// TIA Portal project "sexy pics" (V17)

(* hardware
DEVICE "S7-1200 station_1"  S7-1200 Station
   slot 0: "Rack_0"  S7-1200 Rack  Rack  V1.0
   slot 1: "PLC_1"  CPU 1214C AC/DC/Rly  6ES7 214-1BG40-0XB0  V4.5
DEVICE "HMI_1"  KTP700 Basic PN
   slot 0: "HMI_1"  KTP700 Basic PN  6AV2 123-2GB03-0AX0  17.0.0.0
   slot 1: "HMI_RT_1"  KTP700 Basic PN  6AV2 123-2GB03-0AX0  17.0.0.0
   slot 5: "HMI_1.IE_CP_1"  PROFINET Interface  17.0.0.0
      slot 1: "PROFINET Interface_1"  PROFINET Interface
         slot 1: "Port_1"  Port
*)

// ===== PLC "PLC_1"  CPU 1214C AC/DC/Rly =====

VAR_GLOBAL   // PLC tag table "Default tag table"
   "pbStart" AT %M0.4 : Bool;
   "pbStop" AT %M0.5 : Bool;
   "startTask" AT %M0.0 : Bool;
   "g" AT %M0.1 : Bool;
   "y" AT %M0.2 : Bool;
   "r" AT %M0.3 : Bool;
   "startY" AT %M0.6 : Bool;
   "startR" AT %M0.7 : Bool;
   "reset" AT %M1.0 : Bool;
   "aLow" AT %I0.4 : Bool;
   "aHigh" AT %I0.5 : Bool;
   "wow" AT %M1.1 : Bool;
   "istopper" AT %M1.2 : Bool;
   "digital_In" AT %IW64 : Int;
   "sNorm" AT %MD2 : Real;
   "scaled" AT %MD6 : Real;
   "pbStart2" AT %M1.3 : Bool;
   "pbstop2" AT %M1.4 : Bool;
   "pbStart3" AT %M1.5 : Bool;
   "pbStop3" AT %M1.6 : Bool;
   "halt" AT %M1.7 : Bool;
   "startTask3" AT %M10.0 : Bool;
   "startTask2" AT %M10.1 : Bool;
   "g2" AT %M10.2 : Bool;
   "y2" AT %M10.3 : Bool;
   "r2" AT %M10.4 : Bool;
   "r3" AT %M10.5 : Bool;
   "y3" AT %M10.6 : Bool;
   "inletValveControl" AT %M10.7 : Bool;
   "inletValve" AT %M11.0 : Bool;
   "pbstart5" AT %M11.1 : Bool;
   "pbstop5" AT %M11.2 : Bool;
   "gL" AT %M11.3 : Bool;
   "rR" AT %M11.4 : Bool;
   "yL" AT %M11.5 : Bool;
   "yR" AT %M11.6 : Bool;
   "rL" AT %M11.7 : Bool;
   "gR" AT %M12.0 : Bool;
   "startTask4" AT %M12.1 : Bool;
   "startTask5" AT %M12.2 : Bool;
   "g1" AT %Q0.0 : Bool;
   "y1" AT %Q0.1 : Bool;
   "r1" AT %Q0.2 : Bool;
   "r0" AT %Q0.5 : Bool;
   "y0" AT %Q0.4 : Bool;
   "g0" AT %Q0.3 : Bool;
   "pbStartInput" AT %I0.2 : Bool;
   "pbStartControl" AT %I0.0 : Bool;
   "pbStopControl" AT %I0.1 : Bool;
   "startTaskControl" AT %M12.3 : Bool;
   "aG1" AT %M12.4 : Bool;
   "aY1" AT %M12.5 : Bool;
   "aR1" AT %M12.6 : Bool;
   "aY2" AT %M12.7 : Bool;
   "analogR2" AT %M13.0 : Bool;
   "ag2" AT %M13.1 : Bool;
   "m1Input" AT %MD14 : DInt;
   "m1PT" AT %MD18 : DInt;
   "m1ET" AT %MD22 : DInt;
   "m1CntDown" AT %MD26 : DInt;
   "m1CountUp" AT %MD30 : DInt;
   "m2Input" AT %MD34 : DInt;
   "m2PT" AT %MD38 : DInt;
   "m2ET" AT %MD42 : DInt;
   "m2CntDown" AT %MD46 : DInt;
   "m2CountUp" AT %MD50 : DInt;
   "m3Input" AT %MD54 : DInt;
   "m3PT" AT %MD58 : DInt;
   "m3ET" AT %MD62 : DInt;
   "m3CntDown" AT %MD66 : DInt;
   "m3CountUp" AT %MD70 : DInt;
   "t2_m1Input" AT %MD74 : DInt;
   "t2_m1PT" AT %MD78 : DInt;
   "t2_m1ET" AT %MD82 : DInt;
   "t2_m1CntDown" AT %MD86 : DInt;
   "t2_m1CountUp" AT %MD90 : DInt;
   "t2_m2Input" AT %MD94 : DInt;
   "t2_m2PT" AT %MD98 : DInt;
   "t2_m2ET" AT %MD102 : DInt;
   "t2_m2CntDown" AT %MD106 : DInt;
   "t2_m2CountUp" AT %MD110 : DInt;
   "t2_m3Input" AT %MD114 : DInt;
   "t2_m3PT" AT %MD118 : DInt;
   "t2_m3ET" AT %MD122 : DInt;
   "t2_m3CntDown" AT %MD126 : DInt;
   "t2_m3CountUp" AT %MD130 : DInt;
END_VAR

DATA_BLOCK "Task1_DB"   // DB4
{ S7_Optimized_Access := 'TRUE' }
VERSION : 0.1
// stored: InstanceOfName Task1
"Task1"
BEGIN
END_DATA_BLOCK

DATA_BLOCK "Task1_DB_1"   // DB5
{ S7_Optimized_Access := 'TRUE' }
VERSION : 0.1
// stored: InstanceOfName Task1
"Task1"
BEGIN
END_DATA_BLOCK

DATA_BLOCK "Task1_DB_2"   // DB6
{ S7_Optimized_Access := 'TRUE' }
VERSION : 0.1
// stored: InstanceOfName Task1
"Task1"
BEGIN
END_DATA_BLOCK

DATA_BLOCK "Task2_DB"   // DB8
{ S7_Optimized_Access := 'TRUE' }
VERSION : 0.1
// stored: InstanceOfName Task2
"Task2"
BEGIN
END_DATA_BLOCK

DATA_BLOCK "Task2_DB_1"   // DB9
{ S7_Optimized_Access := 'TRUE' }
VERSION : 0.1
// stored: InstanceOfName Task2
"Task2"
BEGIN
END_DATA_BLOCK

DATA_BLOCK "Task1_DB_3"   // DB10
{ S7_Optimized_Access := 'TRUE' }
VERSION : 0.1
// stored: InstanceOfName Task1
"Task1"
BEGIN
END_DATA_BLOCK

DATA_BLOCK "Task2_DB_2"   // DB11
{ S7_Optimized_Access := 'TRUE' }
VERSION : 0.1
// stored: InstanceOfName Task2
"Task2"
BEGIN
END_DATA_BLOCK

DATA_BLOCK "Task2_DB_3"   // DB12
{ S7_Optimized_Access := 'TRUE' }
VERSION : 0.1
// stored: InstanceOfName Task2
"Task2"
BEGIN
END_DATA_BLOCK

DATA_BLOCK "Task1_DB_4"   // DB17
{ S7_Optimized_Access := 'TRUE' }
VERSION : 0.1
// stored: InstanceOfName Task1
"Task1"
BEGIN
END_DATA_BLOCK

DATA_BLOCK "Task2_DB_4"   // DB18
{ S7_Optimized_Access := 'TRUE' }
VERSION : 0.1
// stored: InstanceOfName Task2
"Task2"
BEGIN
END_DATA_BLOCK

DATA_BLOCK "Task2_DB_5"   // DB19
{ S7_Optimized_Access := 'TRUE' }
VERSION : 0.1
// stored: InstanceOfName Task2
"Task2"
BEGIN
END_DATA_BLOCK

DATA_BLOCK "Task3_DB"   // DB20
{ S7_Optimized_Access := 'TRUE' }
VERSION : 0.1
// stored: InstanceOfName Task3
"Task3"
BEGIN
END_DATA_BLOCK

DATA_BLOCK "task5_DB"   // DB21
{ S7_Optimized_Access := 'TRUE' }
VERSION : 0.1
// stored: InstanceOfName task5
"task5"
BEGIN
END_DATA_BLOCK

DATA_BLOCK "task4_DB"   // DB23
{ S7_Optimized_Access := 'TRUE' }
VERSION : 0.1
// stored: InstanceOfName task4
"task4"
BEGIN
END_DATA_BLOCK

// folder: System blocks/Program resources

DATA_BLOCK "IEC_Timer_0_DB"   // DB1
{ S7_Optimized_Access := 'TRUE' }
AUTHOR : Simatic
FAMILY : IEC
NAME : IEC_TMR
VERSION : 1.0
// stored: InstanceOfName IEC_TIMER
"IEC_TIMER"
BEGIN
END_DATA_BLOCK

DATA_BLOCK "IEC_Timer_0_DB_1"   // DB2
{ S7_Optimized_Access := 'TRUE' }
AUTHOR : Simatic
FAMILY : IEC
NAME : IEC_TMR
VERSION : 1.0
// stored: InstanceOfName IEC_TIMER
"IEC_TIMER"
BEGIN
END_DATA_BLOCK

DATA_BLOCK "IEC_Timer_0_DB_2"   // DB3
{ S7_Optimized_Access := 'TRUE' }
AUTHOR : Simatic
FAMILY : IEC
NAME : IEC_TMR
VERSION : 1.0
// stored: InstanceOfName IEC_TIMER
"IEC_TIMER"
BEGIN
END_DATA_BLOCK

DATA_BLOCK "IEC_Timer_0_DB_3"   // DB7
{ S7_Optimized_Access := 'TRUE' }
AUTHOR : Simatic
FAMILY : IEC
NAME : IEC_TMR
VERSION : 1.0
// stored: InstanceOfName IEC_TIMER
"IEC_TIMER"
BEGIN
END_DATA_BLOCK

DATA_BLOCK "IEC_Timer_0_DB_4"   // DB13
{ S7_Optimized_Access := 'TRUE' }
AUTHOR : Simatic
FAMILY : IEC
NAME : IEC_TMR
VERSION : 1.0
// stored: InstanceOfName IEC_TIMER
"IEC_TIMER"
BEGIN
END_DATA_BLOCK

DATA_BLOCK "LgreenToYellowTimer"   // DB14
{ S7_Optimized_Access := 'TRUE' }
AUTHOR : Simatic
FAMILY : IEC
NAME : IEC_TMR
VERSION : 1.0
// stored: InstanceOfName IEC_TIMER
"IEC_TIMER"
BEGIN
END_DATA_BLOCK

DATA_BLOCK "yellowTimer"   // DB15
{ S7_Optimized_Access := 'TRUE' }
AUTHOR : Simatic
FAMILY : IEC
NAME : IEC_TMR
VERSION : 1.0
// stored: InstanceOfName IEC_TIMER
"IEC_TIMER"
BEGIN
END_DATA_BLOCK

DATA_BLOCK "backToYellowTimer"   // DB16
{ S7_Optimized_Access := 'TRUE' }
AUTHOR : Simatic
FAMILY : IEC
NAME : IEC_TMR
VERSION : 1.0
// stored: InstanceOfName IEC_TIMER
"IEC_TIMER"
BEGIN
END_DATA_BLOCK

DATA_BLOCK "trafficReturnYello"   // DB22
{ S7_Optimized_Access := 'TRUE' }
AUTHOR : Simatic
FAMILY : IEC
NAME : IEC_TMR
VERSION : 1.0
// stored: InstanceOfName IEC_TIMER
"IEC_TIMER"
BEGIN
END_DATA_BLOCK

DATA_BLOCK "IEC_Timer_0_DB_5"   // DB24
{ S7_Optimized_Access := 'TRUE' }
AUTHOR : Simatic
FAMILY : IEC
NAME : IEC_TMR
VERSION : 1.0
// stored: InstanceOfName IEC_TIMER
"IEC_TIMER"
BEGIN
END_DATA_BLOCK

// folder: (top level)

FUNCTION_BLOCK "Task1"   // FB1, LAD
{ S7_Optimized_Access := 'TRUE' }
VERSION : 0.1
   VAR_INPUT
      pbStart : Bool;
      pbStop : Bool;
   END_VAR
   VAR_OUTPUT
      g : Bool;
      r : Bool;
      y : Bool;
      gOut : Bool;
      yOut : Bool;
      rOut : Bool;
   END_VAR
   VAR_TEMP
      m1CountUpddd : DInt;
   END_VAR
BEGIN

REGION Network 1
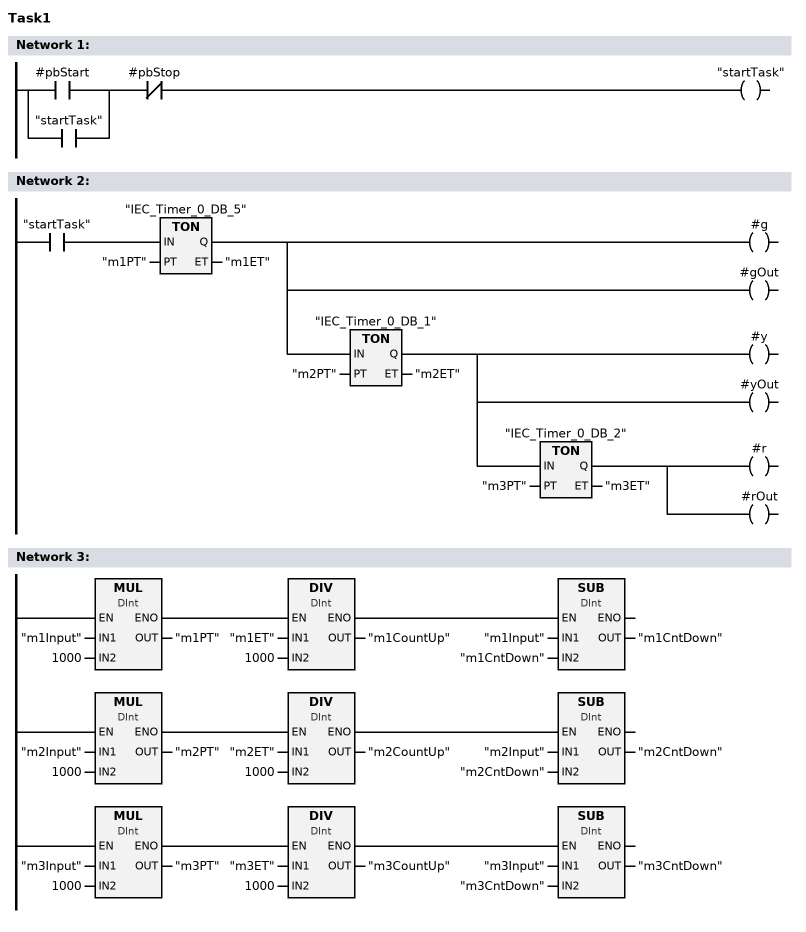
   RUNG wire#powerrail
      Contact( #pbStart )
      wire#w1
      I_Contact( #pbStop )
      Coil( "startTask" )
   END_RUNG
   RUNG wire#powerrail
      Contact( "startTask" )
   END_RUNG wire#w1
   // the same network as SCL:
   "startTask" := (#pbStart OR "startTask") AND NOT #pbStop;
END_REGION

REGION Network 2
   "IEC_Timer_0_DB_5".TON(IN := "startTask", PT := "m1PT", ET => "m1ET");
   #g := "IEC_Timer_0_DB_5".Q;
   #gOut := "IEC_Timer_0_DB_5".Q;
   "IEC_Timer_0_DB_1".TON(IN := "IEC_Timer_0_DB_5".Q, PT := "m2PT", ET => "m2ET");
   #y := "IEC_Timer_0_DB_1".Q;
   #yOut := "IEC_Timer_0_DB_1".Q;
   "IEC_Timer_0_DB_2".TON(IN := "IEC_Timer_0_DB_1".Q, PT := "m3PT", ET => "m3ET");
   #r := "IEC_Timer_0_DB_2".Q;
   #rOut := "IEC_Timer_0_DB_2".Q;
END_REGION

REGION Network 3
   RUNG wire#powerrail
      { S7_Templates := "SrcType := DInt" } Mul(in1 := "m1Input", in2 := 1000, out => "m1PT")
      { S7_Templates := "SrcType := DInt" } Div(in1 := "m1ET", in2 := 1000, out => "m1CountUp")
      { S7_Templates := "SrcType := DInt" } Sub(in1 := "m1Input", in2 := "m1CntDown", out => "m1CntDown")
   END_RUNG
   RUNG wire#powerrail
      { S7_Templates := "SrcType := DInt" } Mul(in1 := "m2Input", in2 := 1000, out => "m2PT")
      { S7_Templates := "SrcType := DInt" } Div(in1 := "m2ET", in2 := 1000, out => "m2CountUp")
      { S7_Templates := "SrcType := DInt" } Sub(in1 := "m2Input", in2 := "m2CntDown", out => "m2CntDown")
   END_RUNG
   RUNG wire#powerrail
      { S7_Templates := "SrcType := DInt" } Mul(in1 := "m3Input", in2 := 1000, out => "m3PT")
      { S7_Templates := "SrcType := DInt" } Div(in1 := "m3ET", in2 := 1000, out => "m3CountUp")
      { S7_Templates := "SrcType := DInt" } Sub(in1 := "m3Input", in2 := "m3CntDown", out => "m3CntDown")
   END_RUNG
   // the same network as SCL:
   "m1PT" := "m1Input" * 1000;
   "m1CountUp" := "m1ET" / 1000;
   "m1CntDown" := "m1Input" - "m1CntDown";
   "m2PT" := "m2Input" * 1000;
   "m2CountUp" := "m2ET" / 1000;
   "m2CntDown" := "m2Input" - "m2CntDown";
   "m3PT" := "m3Input" * 1000;
   "m3CountUp" := "m3ET" / 1000;
   "m3CntDown" := "m3Input" - "m3CntDown";
END_REGION
END_FUNCTION_BLOCK

FUNCTION_BLOCK "Task2"   // FB2, LAD
{ S7_Optimized_Access := 'TRUE' }
VERSION : 0.1
   VAR_INPUT
      pbStart2 : Bool;
      pbStop2 : Bool;
   END_VAR
   VAR_OUTPUT
      g2 : Bool;
      y2 : Bool;
      r2 : Bool;
      yOut : Bool;
      rOut : Bool;
      gOut : Bool;
   END_VAR
   VAR_TEMP   // added for the SCL form of the ladder/FBD networks
      _w1 : Bool;
   END_VAR
BEGIN

REGION Network 1
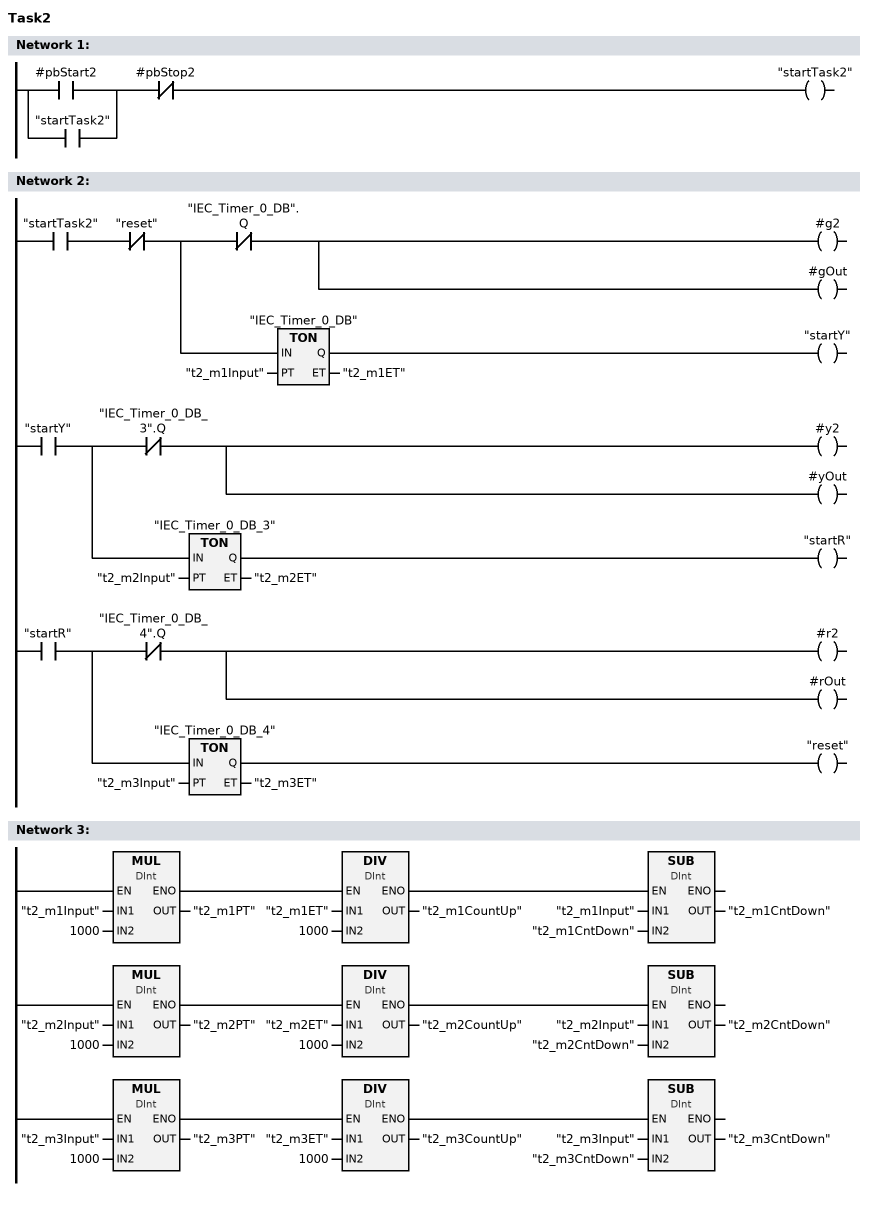
   RUNG wire#powerrail
      Contact( #pbStart2 )
      wire#w1
      I_Contact( #pbStop2 )
      Coil( "startTask2" )
   END_RUNG
   RUNG wire#powerrail
      Contact( "startTask2" )
   END_RUNG wire#w1
   // the same network as SCL:
   "startTask2" := (#pbStart2 OR "startTask2") AND NOT #pbStop2;
END_REGION

REGION Network 2
   #_w1 := "startTask2" AND NOT "reset";
   #g2 := #_w1 AND NOT "IEC_Timer_0_DB".Q;
   #gOut := #g2;
   "IEC_Timer_0_DB".TON(IN := #_w1, PT := "t2_m1Input", ET => "t2_m1ET");
   "startY" := "IEC_Timer_0_DB".Q;
   #y2 := "startY" AND NOT "IEC_Timer_0_DB_3".Q;
   #yOut := #y2;
   "IEC_Timer_0_DB_3".TON(IN := "startY", PT := "t2_m2Input", ET => "t2_m2ET");
   "startR" := "IEC_Timer_0_DB_3".Q;
   #r2 := "startR" AND NOT "IEC_Timer_0_DB_4".Q;
   #rOut := #r2;
   "IEC_Timer_0_DB_4".TON(IN := "startR", PT := "t2_m3Input", ET => "t2_m3ET");
   "reset" := "IEC_Timer_0_DB_4".Q;
END_REGION

REGION Network 3
   RUNG wire#powerrail
      { S7_Templates := "SrcType := DInt" } Mul(in1 := "t2_m1Input", in2 := 1000, out => "t2_m1PT")
      { S7_Templates := "SrcType := DInt" } Div(in1 := "t2_m1ET", in2 := 1000, out => "t2_m1CountUp")
      { S7_Templates := "SrcType := DInt" } Sub(in1 := "t2_m1Input", in2 := "t2_m1CntDown", out => "t2_m1CntDown")
   END_RUNG
   RUNG wire#powerrail
      { S7_Templates := "SrcType := DInt" } Mul(in1 := "t2_m2Input", in2 := 1000, out => "t2_m2PT")
      { S7_Templates := "SrcType := DInt" } Div(in1 := "t2_m2ET", in2 := 1000, out => "t2_m2CountUp")
      { S7_Templates := "SrcType := DInt" } Sub(in1 := "t2_m2Input", in2 := "t2_m2CntDown", out => "t2_m2CntDown")
   END_RUNG
   RUNG wire#powerrail
      { S7_Templates := "SrcType := DInt" } Mul(in1 := "t2_m3Input", in2 := 1000, out => "t2_m3PT")
      { S7_Templates := "SrcType := DInt" } Div(in1 := "t2_m3ET", in2 := 1000, out => "t2_m3CountUp")
      { S7_Templates := "SrcType := DInt" } Sub(in1 := "t2_m3Input", in2 := "t2_m3CntDown", out => "t2_m3CntDown")
   END_RUNG
   // the same network as SCL:
   "t2_m1PT" := "t2_m1Input" * 1000;
   "t2_m1CountUp" := "t2_m1ET" / 1000;
   "t2_m1CntDown" := "t2_m1Input" - "t2_m1CntDown";
   "t2_m2PT" := "t2_m2Input" * 1000;
   "t2_m2CountUp" := "t2_m2ET" / 1000;
   "t2_m2CntDown" := "t2_m2Input" - "t2_m2CntDown";
   "t2_m3PT" := "t2_m3Input" * 1000;
   "t2_m3CountUp" := "t2_m3ET" / 1000;
   "t2_m3CntDown" := "t2_m3Input" - "t2_m3CntDown";
END_REGION
END_FUNCTION_BLOCK

FUNCTION_BLOCK "Task3"   // FB3, LAD
{ S7_Optimized_Access := 'TRUE' }
VERSION : 0.1
   VAR_INPUT
      pbStart3 : Bool;
      pbStop3 : Bool;
      inletValveControl : Bool;
      buttonLow3 : Bool;
   END_VAR
   VAR_OUTPUT
      LLS : Bool;
      inletValve : Bool;
      y3 : Bool;
   END_VAR
   VAR
      Memstarter : Bool;
      Memstopper : Bool;
   END_VAR
BEGIN

REGION Network 1
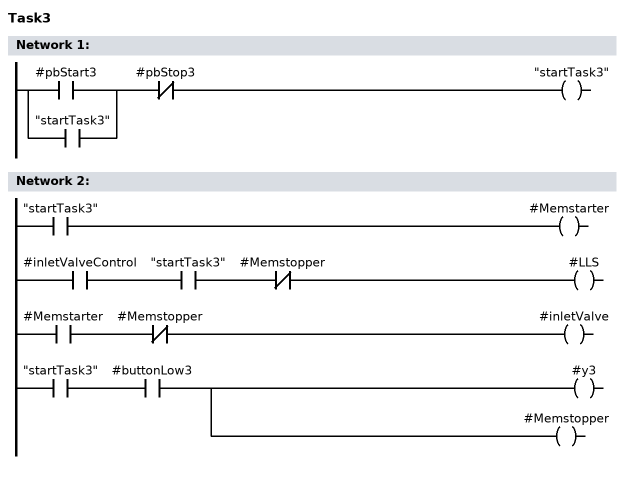
   RUNG wire#powerrail
      Contact( #pbStart3 )
      wire#w1
      I_Contact( #pbStop3 )
      Coil( "startTask3" )
   END_RUNG
   RUNG wire#powerrail
      Contact( "startTask3" )
   END_RUNG wire#w1
   // the same network as SCL:
   "startTask3" := (#pbStart3 OR "startTask3") AND NOT #pbStop3;
END_REGION

REGION Network 2
   RUNG wire#powerrail
      Contact( "startTask3" )
      Coil( #Memstarter )
   END_RUNG
   RUNG wire#powerrail
      Contact( #inletValveControl )
      Contact( "startTask3" )
      I_Contact( #Memstopper )
      Coil( #LLS )
   END_RUNG
   RUNG wire#powerrail
      Contact( #Memstarter )
      I_Contact( #Memstopper )
      Coil( #inletValve )
   END_RUNG
   RUNG wire#powerrail
      Contact( "startTask3" )
      Contact( #buttonLow3 )
      wire#w1
      Coil( #y3 )
   END_RUNG
   RUNG wire#w1
      Coil( #Memstopper )
   END_RUNG
   // the same network as SCL:
   #Memstarter := "startTask3";
   #LLS := #inletValveControl AND "startTask3" AND NOT #Memstopper;
   #inletValve := #Memstarter AND NOT #Memstopper;
   #y3 := "startTask3" AND #buttonLow3;
   #Memstopper := #y3;
END_REGION
END_FUNCTION_BLOCK

FUNCTION_BLOCK "task4"   // FB4, LAD
{ S7_Optimized_Access := 'TRUE' }
VERSION : 0.1
   VAR_INPUT
      pbStart : Bool;
      pbStop : Bool;
   END_VAR
   VAR_OUTPUT
      r : Bool;
      y : Bool;
      g : Bool;
   END_VAR
   VAR_TEMP   // added for the SCL form of the ladder/FBD networks
      _w1 : Bool;
   END_VAR
BEGIN

REGION Network 1
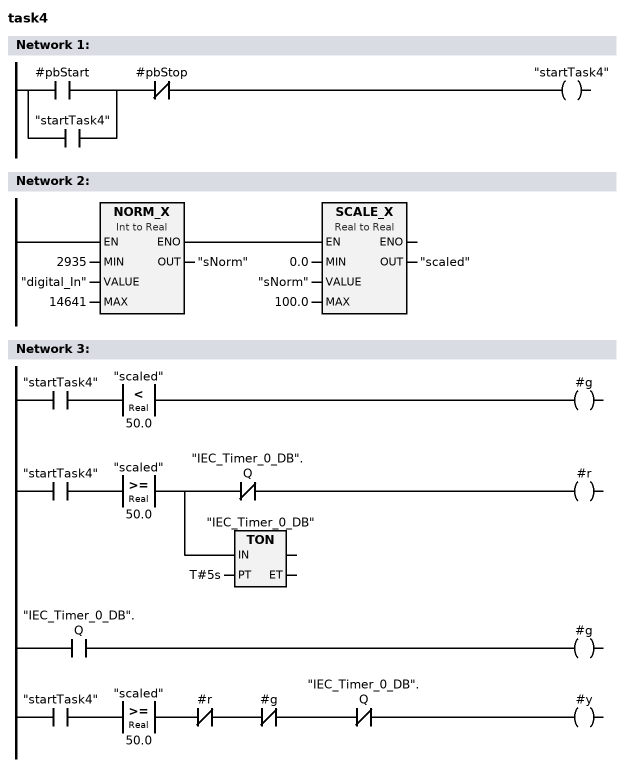
   RUNG wire#powerrail
      Contact( #pbStart )
      wire#w1
      I_Contact( #pbStop )
      Coil( "startTask4" )
   END_RUNG
   RUNG wire#powerrail
      Contact( "startTask4" )
   END_RUNG wire#w1
   // the same network as SCL:
   "startTask4" := (#pbStart OR "startTask4") AND NOT #pbStop;
END_REGION

REGION Network 2
   RUNG wire#powerrail
      { S7_Templates := "[SrcType := Int, DestType := Real]" } Normalize(min := 2935, value := "digital_In", max := 14641, out => "sNorm")
      { S7_Templates := "[SrcType := Real, DestType := Real]" } Scale(min := 0.0, value := "sNorm", max := 100.0, out => "scaled")
   END_RUNG
   // the same network as SCL:
   "sNorm" := NORM_X(MIN := 2935, VALUE := "digital_In", MAX := 14641);
   "scaled" := SCALE_X(MIN := 0.0, VALUE := "sNorm", MAX := 100.0);
END_REGION

REGION Network 3
   #g := "startTask4" AND ("scaled" < 50.0);
   #_w1 := "startTask4" AND ("scaled" >= 50.0);
   #r := #_w1 AND NOT "IEC_Timer_0_DB".Q;
   "IEC_Timer_0_DB".TON(IN := #_w1, PT := T#5s);
   #g := "IEC_Timer_0_DB".Q;
   #y := "startTask4" AND ("scaled" >= 50.0) AND NOT #r AND NOT #g AND NOT "IEC_Timer_0_DB".Q;
END_REGION
END_FUNCTION_BLOCK

FUNCTION_BLOCK "task5"   // FB5, LAD
{ S7_Optimized_Access := 'TRUE' }
VERSION : 0.1
   VAR_INPUT
      pbStart : Bool;
      pbStop : Bool;
   END_VAR
   VAR_OUTPUT
      gL : Bool;
      rR : Bool;
      yL : Bool;
      yR : Bool;
      rL : Bool;
      gR : Bool;
      analog_yL : Bool;
      analog_yR : Bool;
      analog_gL : Bool;
      analog_gR : Bool;
      analog_rL : Bool;
      analog_rR : Bool;
   END_VAR
   VAR
      interlockReturn : Bool;
      toYellow : Bool;
      interlockStopperYellow : Bool;
      returnBackToYellow : Bool;
   END_VAR
   VAR_TEMP   // added for the SCL form of the ladder/FBD networks
      _w1 : Bool;
   END_VAR
BEGIN

REGION Network 1
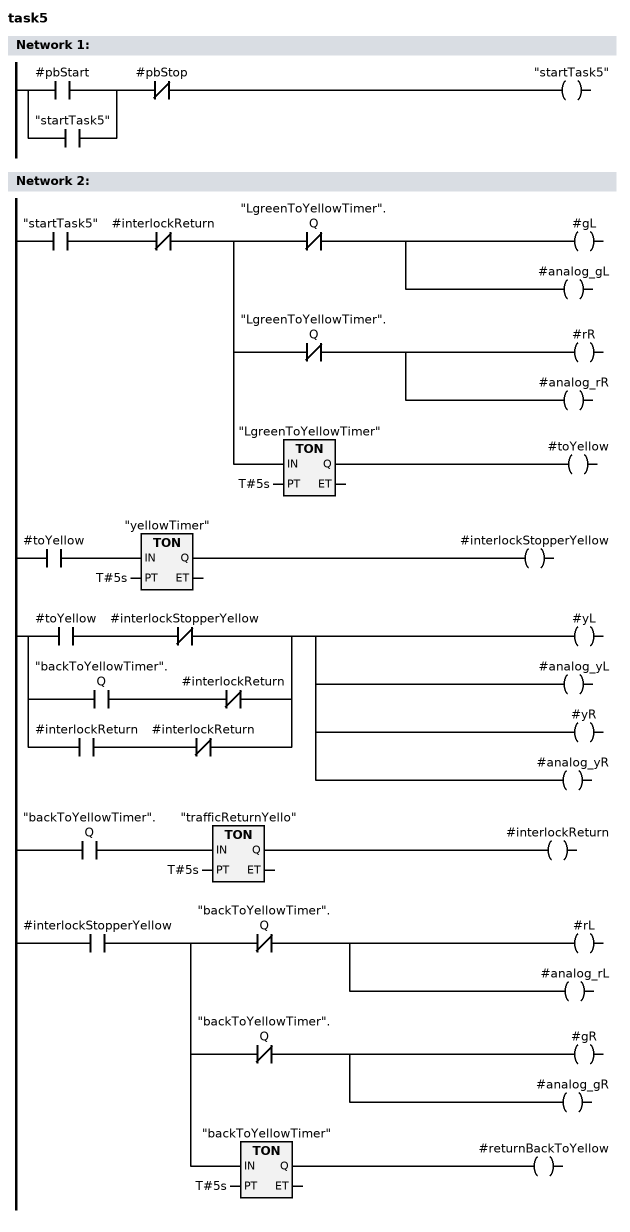
   RUNG wire#powerrail
      Contact( #pbStart )
      wire#w1
      I_Contact( #pbStop )
      Coil( "startTask5" )
   END_RUNG
   RUNG wire#powerrail
      Contact( "startTask5" )
   END_RUNG wire#w1
   // the same network as SCL:
   "startTask5" := (#pbStart OR "startTask5") AND NOT #pbStop;
END_REGION

REGION Network 2
   #_w1 := "startTask5" AND NOT #interlockReturn;
   #gL := #_w1 AND NOT "LgreenToYellowTimer".Q;
   #analog_gL := #gL;
   #rR := #_w1 AND NOT "LgreenToYellowTimer".Q;
   #analog_rR := #rR;
   "LgreenToYellowTimer".TON(IN := #_w1, PT := T#5s);
   #toYellow := "LgreenToYellowTimer".Q;
   "yellowTimer".TON(IN := #toYellow, PT := T#5s);
   #interlockStopperYellow := "yellowTimer".Q;
   #yL := (#toYellow AND NOT #interlockStopperYellow) OR ("backToYellowTimer".Q AND NOT #interlockReturn) OR (#interlockReturn AND NOT #interlockReturn);
   #analog_yL := #yL;
   #yR := #yL;
   #analog_yR := #yL;
   "trafficReturnYello".TON(IN := "backToYellowTimer".Q, PT := T#5s);
   #interlockReturn := "trafficReturnYello".Q;
   #rL := #interlockStopperYellow AND NOT "backToYellowTimer".Q;
   #analog_rL := #rL;
   #gR := #interlockStopperYellow AND NOT "backToYellowTimer".Q;
   #analog_gR := #gR;
   "backToYellowTimer".TON(IN := #interlockStopperYellow, PT := T#5s);
   #returnBackToYellow := "backToYellowTimer".Q;
END_REGION
END_FUNCTION_BLOCK

ORGANIZATION_BLOCK "Main"   // OB1, LAD, ProgramCycle
TITLE = "Main Program Sweep (Cycle)"
{ S7_Optimized_Access := 'TRUE' }
VERSION : 0.1
   VAR_INPUT
      Initial_Call : Bool;   // Initial call of this OB
      Remanence : Bool;   // =True, if remanent data are available
   END_VAR
BEGIN

REGION Network 1
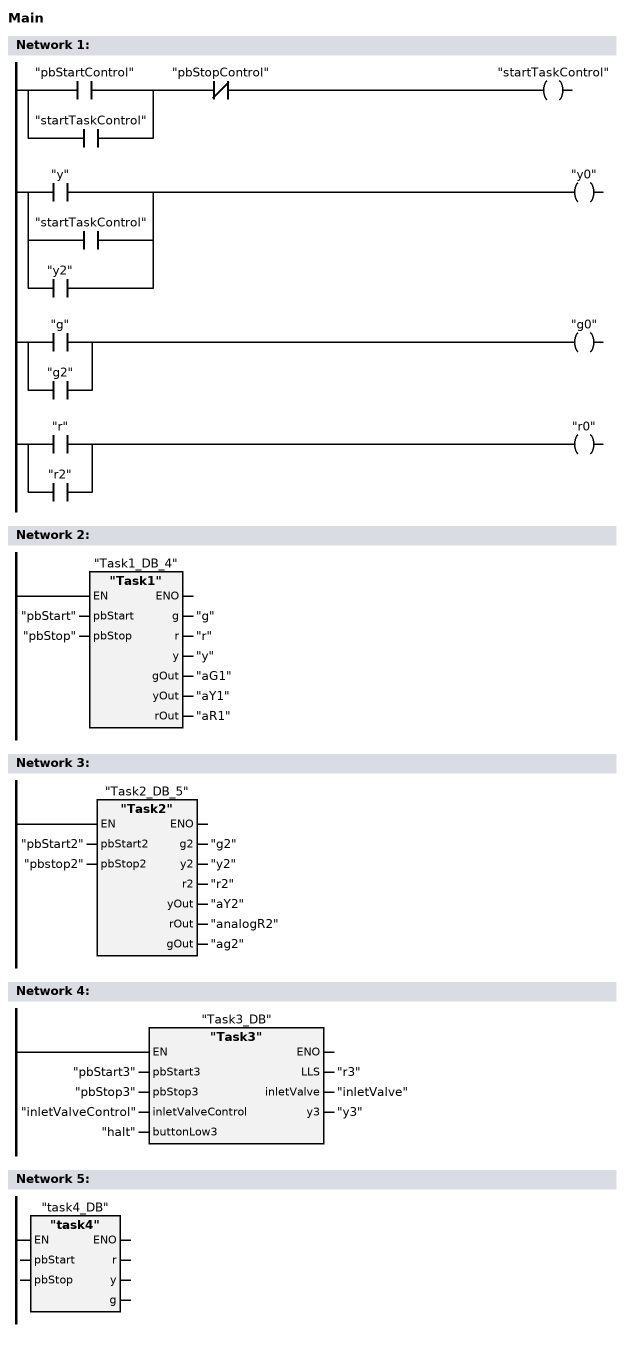
   RUNG wire#powerrail
      Contact( "pbStartControl" )
      wire#w1
      I_Contact( "pbStopControl" )
      Coil( "startTaskControl" )
   END_RUNG
   RUNG wire#powerrail
      Contact( "startTaskControl" )
   END_RUNG wire#w1
   RUNG wire#powerrail
      Contact( "y" )
      wire#w2
      Coil( "y0" )
   END_RUNG
   RUNG wire#powerrail
      Contact( "startTaskControl" )
   END_RUNG wire#w2
   RUNG wire#powerrail
      Contact( "y2" )
   END_RUNG wire#w2
   RUNG wire#powerrail
      Contact( "g" )
      wire#w3
      Coil( "g0" )
   END_RUNG
   RUNG wire#powerrail
      Contact( "g2" )
   END_RUNG wire#w3
   RUNG wire#powerrail
      Contact( "r" )
      wire#w4
      Coil( "r0" )
   END_RUNG
   RUNG wire#powerrail
      Contact( "r2" )
   END_RUNG wire#w4
   // the same network as SCL:
   "startTaskControl" := ("pbStartControl" OR "startTaskControl") AND NOT "pbStopControl";
   "y0" := "y" OR "startTaskControl" OR "y2";
   "g0" := "g" OR "g2";
   "r0" := "r" OR "r2";
END_REGION

REGION Network 2
   RUNG wire#powerrail
      "Task1_DB_4"(pbStart := "pbStart", pbStop := "pbStop", g => "g", r => "r", y => "y", gOut => "aG1", yOut => "aY1", rOut => "aR1")
   END_RUNG
   // the same network as SCL:
   "Task1_DB_4"(pbStart := "pbStart",   // "Task1"
                pbStop := "pbStop",
                g => "g",
                r => "r",
                y => "y",
                gOut => "aG1",
                yOut => "aY1",
                rOut => "aR1");
END_REGION

REGION Network 3
   RUNG wire#powerrail
      "Task2_DB_5"(pbStart2 := "pbStart2", pbStop2 := "pbstop2", g2 => "g2", y2 => "y2", r2 => "r2", yOut => "aY2", rOut => "analogR2", gOut => "ag2")
   END_RUNG
   // the same network as SCL:
   "Task2_DB_5"(pbStart2 := "pbStart2",   // "Task2"
                pbStop2 := "pbstop2",
                g2 => "g2",
                y2 => "y2",
                r2 => "r2",
                yOut => "aY2",
                rOut => "analogR2",
                gOut => "ag2");
END_REGION

REGION Network 4
   RUNG wire#powerrail
      "Task3_DB"(pbStart3 := "pbStart3", pbStop3 := "pbStop3", inletValveControl := "inletValveControl", buttonLow3 := "halt", LLS => "r3", inletValve => "inletValve", y3 => "y3")
   END_RUNG
   // the same network as SCL:
   "Task3_DB"(pbStart3 := "pbStart3",   // "Task3"
              pbStop3 := "pbStop3",
              inletValveControl := "inletValveControl",
              buttonLow3 := "halt",
              LLS => "r3",
              inletValve => "inletValve",
              y3 => "y3");
END_REGION

REGION Network 5
   RUNG wire#powerrail
      "task4_DB"(pbStart :=, pbStop :=, r =>, y =>, g =>)
   END_RUNG
   // the same network as SCL:
   "task4_DB"();   // "task4"
END_REGION
END_ORGANIZATION_BLOCK

(* ===== HMI "HMI_RT_1" =====
system functions are stored by id; their names below are inferred from use
connection "HMI_Connection_1": ETHERNET, SMART_S7_1200_OMS

HMI tags "Default tag table"
   "pbStart" : Bool = PLC pbStart AT %M0.4, 1 s
   "pbStop" : Bool = PLC pbStop AT %M0.5, 1 s
   "g" : Bool = PLC g AT %M0.1, 1 s
   "y" : Bool = PLC y AT %M0.2, 1 s
   "r" : Bool = PLC r AT %M0.3, 1 s
   "pbStart2" : Bool = PLC pbStart2 AT %M1.3, 1 s
   "halt" : Bool = PLC halt AT %M1.7, 1 s
   "pbStart3" : Bool = PLC pbStart3 AT %M1.5, 1 s
   "pbStop3" : Bool = PLC pbStop3 AT %M1.6, 1 s
   "pbstop2" : Bool = PLC pbstop2 AT %M1.4, 1 s
   "g2" : Bool = PLC g2 AT %M10.2, 1 s
   "y2" : Bool = PLC y2 AT %M10.3, 1 s
   "r3" : Bool = PLC r3 AT %M10.5, 1 s
   "y3" : Bool = PLC y3 AT %M10.6, 1 s
   "inletValve" : Bool = PLC inletValve AT %M11.0, 1 s
   "r2" : Bool = PLC r2 AT %M10.4, 1 s
   "yL" : Bool = PLC yL AT %M11.5, 1 s
   "gL" : Bool = PLC gL AT %M11.3, 1 s
   "rL" : Bool = PLC rL AT %M11.7, 1 s
   "rR" : Bool = PLC rR AT %M11.4, 1 s
   "yR" : Bool = PLC yR AT %M11.6, 1 s
   "gR" : Bool = PLC gR AT %M12.0, 1 s
   "aHigh" : Bool = PLC aHigh AT %I0.5, 1 s
   "pbstart5" : Bool = PLC pbstart5 AT %M11.1, 1 s
   "pbstop5" : Bool = PLC pbstop5 AT %M11.2, 1 s
   "m1Input" : DInt = PLC m1Input AT %MD14, 1 s
   "m2Input" : DInt = PLC m2Input AT %MD34, 1 s
   "m1CntDown" : DInt = PLC m1CntDown AT %MD26, 1 s
   "m1CountUp" : DInt = PLC m1CountUp AT %MD30, 1 s
   "m2CntDown" : DInt = PLC m2CntDown AT %MD46, 1 s
   "m2CountUp" : DInt = PLC m2CountUp AT %MD50, 1 s
   "m3Input" : DInt = PLC m3Input AT %MD54, 1 s
   "m3CntDown" : DInt = PLC m3CntDown AT %MD66, 1 s
   "m3CountUp" : DInt = PLC m3CountUp AT %MD70, 1 s
   "t2_m1Input" : DInt = PLC t2_m1Input AT %MD74, 1 s
   "t2_m2Input" : DInt = PLC t2_m2Input AT %MD94, 1 s
   "t2_m3Input" : DInt = PLC t2_m3Input AT %MD114, 1 s
   "t2_m1CntDown" : DInt = PLC t2_m1CntDown AT %MD86, 1 s
   "t2_m1CountUp" : DInt = PLC t2_m1CountUp AT %MD90, 1 s
   "t2_m2CntDown" : DInt = PLC t2_m2CntDown AT %MD106, 1 s
   "t2_m2CountUp" : DInt = PLC t2_m2CountUp AT %MD110, 1 s
   "t2_m3CntDown" : DInt = PLC t2_m3CntDown AT %MD126, 1 s
   "t2_m3CountUp" : DInt = PLC t2_m3CountUp AT %MD130, 1 s
   "scaled" : Real = PLC scaled AT %MD6, 1 s

screen "Root screen" 800x480, template "Template_1"
   GraphicView "Graphic view_1" at 18,20 size 84x84; Picture "275542019_5352027011475781_8646763153125628757_n"
   TextField "Text field_1" at 111,20 size 617x37; Text 'PLC TRAINING COMPILATION OF PROJECTS'
   TextField "Text field_2" at 111,64 size 173x25; Text 'BY: NICO GUARNES'
   Button "Button_1" at 54,156 size 212x100; TextOff 'PRACTICAL 1: Motor Control'
      on Release: ActivateScreen("Practical_1", 0)
   Button "Button_2" at 299,156 size 212x100; TextOff 'PRACTICAL 2: Sequential Motor Control'
      on Release: ActivateScreen("Practical_2", 0)
   Button "Button_3" at 546,156 size 212x100; TextOff 'PRACTICAL 3: Control Level of a Single Tank'
      on Release: ActivateScreen("Practical_3", 0)
   Button "Button_4" at 50,290 size 212x100; TextOff 'PRACTICAL 4: Control Mixing in a Tank'
      on Release: ActivateScreen("Practical_4", 0)
   Button "Button_5" at 299,290 size 212x100; TextOff 'PRACTICAL 5: Traffic Lights'
      on Release: ActivateScreen("Practical_5", 0)

screen "Practical_1" 800x480, template "Template_1"
   GraphicView "Graphic view_1" at 18,20 size 84x84; Picture "275542019_5352027011475781_8646763153125628757_n"
   TextField "Text field_1" at 111,20 size 455x37; Text 'PRACTICAL 1 : MOTOR CONTROL'
   TextField "Text field_2" at 111,64 size 173x25; Text 'BY: NICO GUARNES'
   Button "Button_1" at 715,41 size 54x48; TextOff 'Text'; PictureOff "home_64dp_FFBE33_FILL1_wght400_GRAD0_opsz48"
      on Release: ActivateScreen("Root screen", 0); ResetBit("pbStop")
      on Press: SetBit("pbStop")
   Button "Button_2" at 11,431 size 96x32; TextOff 'START'
      on Release: ResetBit("pbStart")
      on Press: SetBit("pbStart")
   Button "Button_3" at 123,431 size 96x32; TextOff 'STOP'
      on Press: SetBit("pbStop")
      on Release: ResetBit("pbStop")
   GraphicView "Graphic view_2" at 58,159 size 187x105; Picture "Graphic_3"
      Visibility <- "g"
   GraphicView "Graphic view_3" at 58,159 size 187x105; Picture "Graphic_4"
      Visibility <- "g"
   GraphicView "Graphic view_4" at 308,161 size 187x105; Picture "Graphic_3"
      Visibility <- "y"
   GraphicView "Graphic view_6" at 540,161 size 187x105; Picture "Graphic_3"
      Visibility <- "r"
   GraphicView "Graphic view_5" at 308,161 size 187x105; Picture "Graphic_5"
      Visibility <- "y"
   GraphicView "Graphic view_7" at 540,161 size 187x105; Picture "Graphic_6"
      Visibility <- "r"
   TextField "Text field_11" at 64,138 size 56x17; Text 'MOTOR 1'
   TextField "Text field_3" at 322,134 size 56x17; Text 'MOTOR 1'
   TextField "Text field_4" at 580,130 size 56x17; Text 'MOTOR 3'
   IOField "I/O field_1" at 69,282 size 96x32; FormatPattern 999
      ProcessValue <- "m1Input"
   IOField "I/O field_4" at 69,324 size 96x32; FormatPattern 999
      ProcessValue <- "m1CntDown"
   IOField "I/O field_5" at 69,366 size 96x32; FormatPattern 999
      ProcessValue <- "m1CountUp"
   IOField "I/O field_2" at 323,282 size 96x32; FormatPattern 999
      ProcessValue <- "m2Input"
   IOField "I/O field_3" at 323,324 size 96x32; FormatPattern 999
      ProcessValue <- "m2CntDown"
   IOField "I/O field_6" at 323,366 size 96x32; FormatPattern 999
      ProcessValue <- "m2CountUp"
   IOField "I/O field_7" at 563,282 size 96x32; FormatPattern 999
      ProcessValue <- "m3Input"
   IOField "I/O field_8" at 563,324 size 96x32; FormatPattern 999
      ProcessValue <- "m3CntDown"
   IOField "I/O field_9" at 563,366 size 96x32; FormatPattern 999
      ProcessValue <- "m3CountUp"
   TextField "Text field_5" at 168,332 size 72x17; Text 'Count Down'
   TextField "Text field_6" at 167,373 size 56x17; Text 'Count Up'
   TextField "Text field_7" at 172,290 size 92x17; Text 'Preset Time (s)'
   TextField "Text field_8" at 422,332 size 72x17; Text 'Count Down'
   TextField "Text field_9" at 421,373 size 56x17; Text 'Count Up'
   TextField "Text field_10" at 426,290 size 92x17; Text 'Preset Time (s)'
   TextField "Text field_12" at 676,332 size 72x17; Text 'Count Down'
   TextField "Text field_13" at 675,373 size 56x17; Text 'Count Up'
   TextField "Text field_14" at 680,290 size 92x17; Text 'Preset Time (s)'

screen "Practical_2" 800x480, template "Template_1"
   GraphicView "Graphic view_1" at 18,20 size 84x84; Picture "275542019_5352027011475781_8646763153125628757_n"
   TextField "Text field_1" at 111,20 size 582x34; Text 'PRACTICAL 2 : SEQUENTIAL MOTOR CONTROL'
   TextField "Text field_2" at 111,56 size 173x25; Text 'BY: NICO GUARNES'
   Button "Button_1" at 715,41 size 54x48; TextOff 'Text'; PictureOff "home_64dp_FFBE33_FILL1_wght400_GRAD0_opsz48"
      on Release: ActivateScreen("Root screen", 0); ResetBit("pbstop2")
      on Press: SetBit("pbstop2")
   Button "Button_2" at 11,431 size 96x32; TextOff 'START'
      on Release: ResetBit("pbStart2")
      on Press: SetBit("pbStart2")
   Button "Button_3" at 123,431 size 96x32; TextOff 'STOP'
      on Release: ResetBit("pbstop2")
      on Press: SetBit("pbstop2")
   GraphicView "Graphic view_2" at 58,181 size 187x105; Picture "Graphic_3"
   GraphicView "Graphic view_3" at 58,181 size 187x105; Picture "Graphic_4"
      Visibility <- "g2"
   GraphicView "Graphic view_4" at 280,181 size 187x105; Picture "Graphic_3"
   GraphicView "Graphic view_6" at 518,188 size 187x105; Picture "Graphic_3"
   GraphicView "Graphic view_5" at 280,181 size 187x105; Picture "Graphic_5"
      Visibility <- "y2"
   GraphicView "Graphic view_7" at 518,188 size 187x105; Picture "Graphic_6"
      Visibility <- "r2"
   TextField "Text field_11" at 64,156 size 56x17; Text 'MOTOR 1'
   TextField "Text field_3" at 280,156 size 56x17; Text 'MOTOR 2'
   TextField "Text field_4" at 518,163 size 56x17; Text 'MOTOR 3'
   IOField "I/O field_1" at 65,310 size 96x32; FormatPattern 999
      ProcessValue <- "t2_m1Input"
   IOField "I/O field_4" at 65,352 size 96x32; FormatPattern 999
      ProcessValue <- "t2_m1CntDown"
   IOField "I/O field_5" at 65,394 size 96x32; FormatPattern 999
      ProcessValue <- "t2_m1CountUp"
   IOField "I/O field_2" at 295,310 size 96x32; FormatPattern 999
      ProcessValue <- "t2_m2Input"
   IOField "I/O field_3" at 295,352 size 96x32; FormatPattern 999
      ProcessValue <- "t2_m2CntDown"
   IOField "I/O field_6" at 295,394 size 96x32; FormatPattern 999
      ProcessValue <- "t2_m2CountUp"
   IOField "I/O field_7" at 525,310 size 96x32; FormatPattern 999
      ProcessValue <- "t2_m3Input"
   IOField "I/O field_8" at 525,352 size 96x32; FormatPattern 999
      ProcessValue <- "t2_m3CntDown"
   IOField "I/O field_9" at 525,394 size 96x32; FormatPattern 999
      ProcessValue <- "t2_m3CountUp"
   TextField "Text field_5" at 166,361 size 72x17; Text 'Count Down'
   TextField "Text field_6" at 165,402 size 56x17; Text 'Count Up'
   TextField "Text field_7" at 170,319 size 92x17; Text 'Preset Time (s)'
   TextField "Text field_8" at 402,361 size 72x17; Text 'Count Down'
   TextField "Text field_9" at 403,402 size 56x17; Text 'Count Up'
   TextField "Text field_10" at 402,319 size 92x17; Text 'Preset Time (s)'
   TextField "Text field_12" at 628,361 size 72x17; Text 'Count Down'
   TextField "Text field_13" at 625,402 size 56x17; Text 'Count Up'
   TextField "Text field_14" at 626,319 size 92x17; Text 'Preset Time (s)'

screen "Practical_3" 800x480, template "Template_1"
   GraphicView "Graphic view_1" at 18,20 size 84x84; Picture "275542019_5352027011475781_8646763153125628757_n"
   TextField "Text field_1" at 111,20 size 574x34; Text 'PRACTICAL 3 : SINGLE TANK CONTROL LEVEL'
   TextField "Text field_2" at 111,64 size 173x25; Text 'BY: NICO GUARNES'
   Button "Button_1" at 715,41 size 54x48; TextOff 'Text'; PictureOff "home_64dp_FFBE33_FILL1_wght400_GRAD0_opsz48"
      on Release: ActivateScreen("Root screen", 0)
   Button "Button_2" at 15,151 size 96x32; TextOff 'START'
      on Release: ResetBit("pbStart3")
      on Press: SetBit("pbStart3")
   Button "Button_3" at 15,203 size 96x32; TextOff 'STOP'
      on Release: ResetBit("pbStop3")
      on Press: SetBit("pbStop3")
   GraphicView "Graphic view_5" at 497,432 size 125x38; Picture "Graphic_13"
   GraphicView "Graphic view_10" at 464,432 size 34x38; Picture "Graphic_21"
   GraphicView "Graphic view_9" at 464,397 size 34x38; Picture "Graphic_18"
   GraphicView "Graphic view_4" at 222,144 size 126x34; Picture "Graphic_13"
   GraphicView "Graphic view_6" at 243,140 size 43x36; Picture "Graphic_19"
   GraphicView "Graphic view_2" at 344,143 size 39x36; Picture "Graphic_16"
   GraphicView "Graphic view_8" at 345,177 size 38x55; Picture "Graphic_18"
   GraphicView "Graphic view_7" at 547,431 size 43x36; Picture "Graphic_19"
   GraphicView "Graphic view_3" at 332,203 size 190x208; Picture "Graphic_11"
   Circle "Circle_1" at 351,226 size 25x25
      Appearance <- "y3"
   Circle "Circle_2" at 356,368 size 25x25
      Appearance <- "r3"
   TextField "Text field_3" at 292,227 size 38x25; Text 'LLH'
   TextField "Text field_4" at 297,367 size 36x25; Text 'LLS'
   GraphicView "Graphic view_11" at 244,140 size 43x36; Picture "Graphic_22"
      Visibility <- "inletValve"
   GraphicView "Graphic view_12" at 547,431 size 43x36; Picture "Graphic_23"
      Visibility <- "y3"
   TextField "Text field_11" at 544,414 size 84x17; Text 'OUTLET VALVE'
   TextField "Text field_5" at 222,124 size 73x17; Text 'INLET VALVE'
   Bar "Bar_1" at 206,203 size 80x212; MinimumValue 0; MaximumValue 100

screen "Practical_4" 800x480, template "Template_1"
   GraphicView "Graphic view_16" at 409,434 size 97x26; Picture "Graphic_13"
   GraphicView "Graphic view_17" at 465,431 size 33x28; Picture "Graphic_19"
   GraphicView "Graphic view_18" at 465,431 size 33x28; Picture "Graphic_22"
      Visibility <- "inletValve"
   GraphicView "Graphic view_19" at 376,435 size 35x24; Picture "Graphic_21"
   GraphicView "Graphic view_20" at 376,399 size 34x40; Picture "Graphic_18"
   TextField "Text field_10" at 524,437 size 97x17; Text 'MIXED PRODUCT'
   TextField "Text field_11" at 448,460 size 84x17; Text 'OUTLET VALVE'
   GraphicView "Graphic view_6" at 252,91 size 97x26; Picture "Graphic_13"
   GraphicView "Graphic view_7" at 268,88 size 33x28; Picture "Graphic_19"
   GraphicView "Graphic view_8" at 346,90 size 30x28; Picture "Graphic_16"
   GraphicView "Graphic view_11" at 269,88 size 33x28; Picture "Graphic_22"
      Visibility <- "inletValve"
   GraphicView "Graphic view_10" at 345,114 size 32x32; Picture "Graphic_18"
   GraphicView "Graphic view_9" at 447,92 size 97x26; Picture "Graphic_13"
   GraphicView "Graphic view_12" at 503,90 size 33x28; Picture "Graphic_19"
   GraphicView "Graphic view_13" at 503,90 size 33x28; Picture "Graphic_22"
      Visibility <- "inletValve"
   GraphicView "Graphic view_15" at 415,114 size 32x32; Picture "Graphic_18"
   GraphicView "Graphic view_14" at 415,91 size 33x29; Picture "Graphic_30"
   TextField "Text field_3" at 171,96 size 74x17; Text 'MATERIAL A'
   TextField "Text field_4" at 558,95 size 73x17; Text 'MATERIAL B'
   TextField "Text field_5" at 252,118 size 83x17; Text 'INLET VALVE 1'
   TextField "Text field_6" at 466,115 size 83x17; Text 'INLET VALVE 2'
   GraphicView "Graphic view_1" at 42,20 size 54x58; Picture "275542019_5352027011475781_8646763153125628757_n"
   TextField "Text field_1" at 111,20 size 604x37; Text 'PRACTICAL 4: CONTROL MIXING IN A TANK'
   TextField "Text field_2" at 111,52 size 173x25; Text 'BY: NICO GUARNES'
   Button "Button_1" at 715,41 size 54x48; TextOff 'Text'; PictureOff "home_64dp_FFBE33_FILL1_wght400_GRAD0_opsz48"
      on Release: ActivateScreen("Root screen", 0)
   Button "Button_2" at 15,155 size 96x32; TextOff 'START'
      on Release: ResetBit("pbStart")
      on Press: SetBit("pbStart")
   Button "Button_3" at 15,199 size 96x32; TextOff 'STOP'
      on Release: SetBit("pbStop")
      on Press: SetBit("pbStop")
   GraphicView "Graphic view_3" at 354,188 size 115x161; Picture "Graphic_28"
   GraphicView "Graphic view_2" at 300,137 size 185x297; Picture "Graphic_26"
   GraphicView "Graphic view_4" at 358,178 size 64x154; Picture "Graphic_24"
   GraphicView "Graphic view_5" at 358,178 size 64x154; Picture "Graphic_25"
   TextField "Text field_7" at 494,183 size 107x17; Text 'MATERIAL B LEVEL'
   TextField "Text field_8" at 494,317 size 108x17; Text 'MATERIAL A LEVEL'
   TextField "Text field_9" at 377,355 size 24x17; Text 'LLS'
   Bar "Bar_1" at 227,177 size 64x162; MinimumValue 0; MaximumValue 100
      ProcessValue <- "scaled"
   IOField "I/O field_1" at 226,135 size 66x36; FormatPattern 99999
      ProcessValue <- "scaled"

screen "Practical_5" 800x480, template "Template_1"
   GraphicView "Graphic view_2" at 0,92 size 799x388; Picture "ChatGPT Image Apr 20, 2026, 03_55_33 PM"
   GraphicView "Graphic view_1" at 18,20 size 54x54; Picture "275542019_5352027011475781_8646763153125628757_n"
   TextField "Text field_1" at 111,20 size 432x37; Text 'PRACTICAL 5: TRAFFIC LIGHTS'
   TextField "Text field_2" at 111,50 size 173x25; Text 'BY: NICO GUARNES'
   Button "Button_1" at 715,41 size 54x48; TextOff 'Text'; PictureOff "home_64dp_FFBE33_FILL1_wght400_GRAD0_opsz48"
      on Release: ActivateScreen("Root screen", 0)
   Button "Button_2" at 11,431 size 96x32; TextOff 'START'
      on Release: ResetBit("pbstart5")
      on Press: SetBit("pbstart5")
   Button "Button_3" at 123,431 size 96x32; TextOff 'STOP'
      on Release: ResetBit("pbstop5")
      on Press: SetBit("pbstop5")
   GraphicView "Graphic view_3" at 310,92 size 70x70; Picture "ambulance-paramedic-top-view-design-free-vector-removebg-preview"
   GraphicView "Graphic view_4" at 189,279 size 62x30; Picture "orange - Copy"
   GraphicView "Graphic view_5" at 406,360 size 32x64; Picture "grey"
   GraphicView "Graphic view_6" at 436,410 size 39x70; Picture "blu"
   GraphicView "Graphic view_7" at 550,202 size 68x30; Picture "barney - Copy"
   GraphicView "Graphic view_8" at 275,119 size 64x104; Picture "Tlights"
   GraphicView "Graphic view_9" at 277,306 size 64x104; Picture "Tlights"
   GraphicView "Graphic view_10" at 468,116 size 64x104; Picture "Tlights"
   GraphicView "Graphic view_11" at 470,302 size 64x104; Picture "Tlights"
   Ellipse "Ellipse_3" at 294,177 size 23x24
      Appearance <- "gL"
   Ellipse "Ellipse_1" at 294,152 size 23x24
      Appearance <- "yL"
   Ellipse "Ellipse_2" at 294,129 size 23x24
      Appearance <- "rL"
   Ellipse "Ellipse_13" at 490,362 size 23x24
      Appearance <- "gR"
   Ellipse "Ellipse_14" at 490,337 size 23x24
      Appearance <- "yR"
   Ellipse "Ellipse_15" at 490,314 size 23x24
      Appearance <- "rR"
   Ellipse "Ellipse_4" at 488,176 size 23x24
      Appearance <- "gL"
   Ellipse "Ellipse_5" at 488,151 size 23x24
      Appearance <- "yL"
   Ellipse "Ellipse_6" at 488,128 size 23x24
      Appearance <- "rL"
   Ellipse "Ellipse_16" at 297,364 size 23x24
      Appearance <- "gR"
   Ellipse "Ellipse_17" at 297,339 size 23x24
      Appearance <- "yR"
   Ellipse "Ellipse_18" at 297,316 size 23x24
      Appearance <- "rR"
*)